{attribute addProperty BoxType "EL7041-0000-0018"}
{attribute addProperty Id "ENC_Status_compactAT %I*ENC_Status_compact_58C6E2B94860STM_StatusAT %I*STM_Status_C2B0CAE11620ENC_Control_compactAT %Q*ENC_Control_compact_03701F333240STM_ControlAT %Q*STM_Control_6F24B2C41620STM_VelocityAT %Q*STM_Velocity_1D89B5C21620WcStateAT %I*WcState_F855686C1620InfoDataAT %I*InfoData_1C46E3E796120"}
{attribute addProperty CRC "131180535"}
{attribute addProperty SizeInBites "240"}
{attribute addProperty SizeInBytes "30"}
TYPE EL7041_034F0A8C :
STRUCT
	{attribute addProperty Name "ENC_Status_compact"}
	ENC_Status_compact : ENC_Status_compact_58C6E2B9;
	{attribute addProperty Name "STM_Status"}
	STM_Status : STM_Status_C2B0CAE1;
	{attribute addProperty Name "ENC_Control_compact"}
	ENC_Control_compact : ENC_Control_compact_03701F33;
	{attribute addProperty Name "STM_Control"}
	STM_Control : STM_Control_6F24B2C4;
	{attribute addProperty Name "STM_Velocity"}
	STM_Velocity : STM_Velocity_1D89B5C2;
	{attribute addProperty Name "WcState"}
	WcState : WcState_F855686C;
	{attribute addProperty Name "InfoData"}
	InfoData : InfoData_1C46E3E7;
END_STRUCT
END_TYPE

(* stored: Version 1.2.0.0, ProductVersion 3.1.4024.9
   DUT EL7041_034F0A8C: Id {a87f6df2-bbe3-4af0-9a6d-7f59c0e0b105} *)
